{attribute 'qualified_only'}
VAR_GLOBAL
	monitorValue : UDINT;
	monitorReal	: LREAL;
END_VAR

(* stored: Version 1.1.0.1
   GVL GVL: Id {dc6cc913-77c0-41ef-92a3-2b36cf1d4bae} *)
